(* PLC project Sin nombre, Desconocido Sin nombre 1 *)
(* stored: creationDateTime 2024-11-28T09:53:41, modificationDateTime 2024-12-06T04:11:27 *)

PROGRAM Dimmer
  VAR
    Control_button AT %IX0.0 : BOOL;  (* Push button input *)
    Light_output AT %QX0.0 : BOOL;  (* Light dimmer control output *)
  END_VAR
  VAR
    Light_bright : INT;  (* Step sequence count indicates the bright level *)
    Pulse_regulator : TIME;  (* Value in time of pulse width *)
    Light_on_state : BOOL;  (* Indicates that light is on *)
    Reset_state : BOOL;  (* Reset de counter, change the state to zero *)
    Flag_cicle : BOOL;  (* Flag active during a cicle, 10ms, used to restart *)
    Full_bright : BOOL;  (* Indicates maximum bright, turn the light on directly *)
    CTU0 : CTU;  (* States counter *)
    TP0 : TP;  (* Pulse generator and width corrector *)
    TOF0 : TOF;  (* Cicle generator timer *)
  END_VAR
  VAR  (* added by the conversion: wires and edge detectors of the diagram *)
    R_TRIG1 : R_TRIG;
    R_TRIG2 : R_TRIG;
  END_VAR

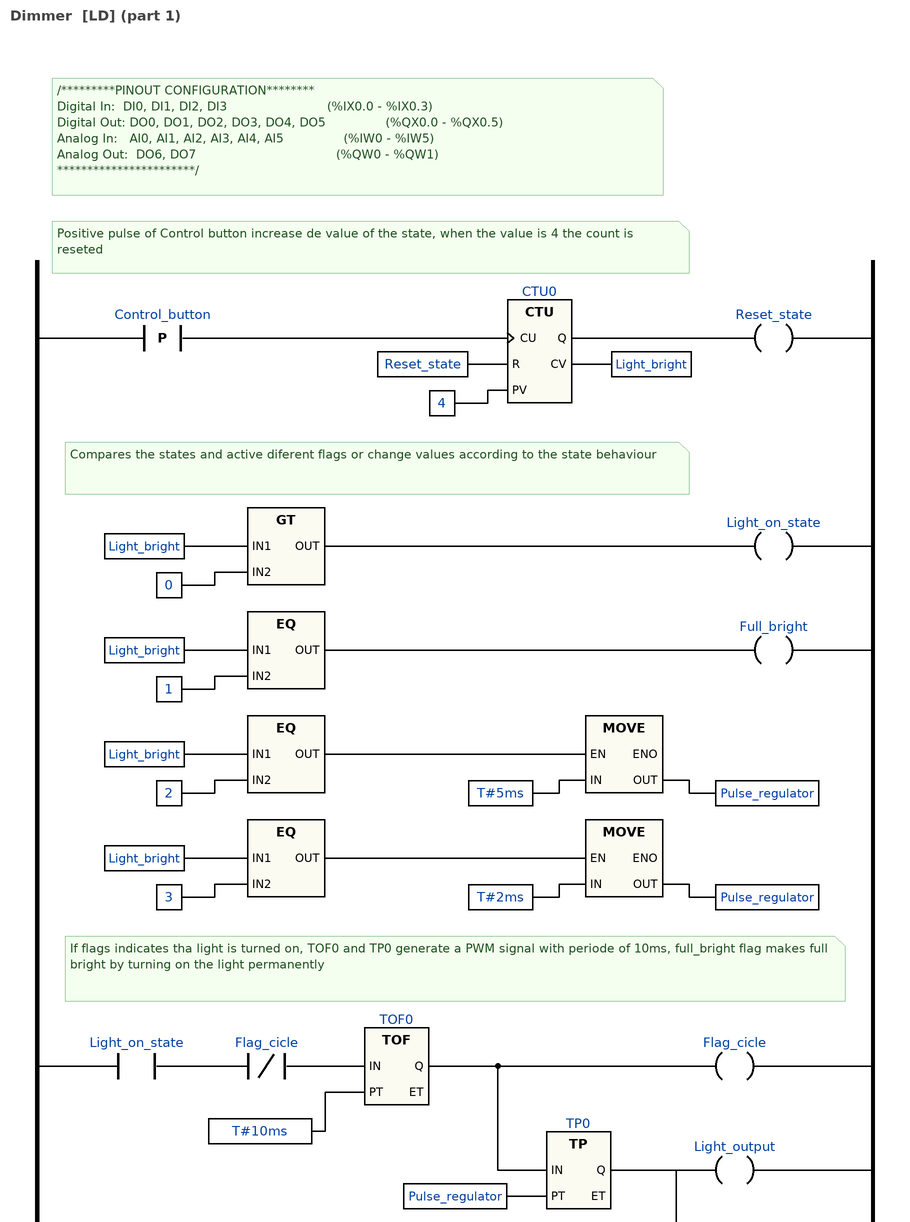
(* LD diagram, written out as Structured Text *)
(* /*********PINOUT CONFIGURATION********
Digital In:  DI0, DI1, DI2, DI3                         (%IX0.0 - %IX0.3)
Digital Out: DO0, DO1, DO2, DO3, DO4, DO5               (%QX0.0 - %QX0.5)
Analog In:   AI0, AI1, AI2, AI3, AI4, AI5               (%IW0 - %IW5)
Analog Out:  DO6, DO7                                   (%QW0 - %QW1)
***********************/ *)
(* Positive pulse of Control button increase de value of the state, when the value is 4 the count is reseted *)
R_TRIG1(CLK := Control_button);
R_TRIG2(CLK := R_TRIG1.Q);
CTU0(CU := R_TRIG2.Q, R := Reset_state, PV := 4);
Reset_state := CTU0.Q;
Light_bright := CTU0.CV;
(* Compares the states and active diferent flags or change values according to the state behaviour *)
(* If flags indicates tha light is turned on, TOF0 and TP0 generate a PWM signal with periode of 10ms, full_bright flag makes full bright by turning on the light permanently *)
TOF0(IN := Light_on_state AND NOT Flag_cicle, PT := T#10ms);
TP0(IN := TOF0.Q, PT := Pulse_regulator);
Light_output := TP0.Q OR Full_bright;
IF Light_bright = 2 THEN Pulse_regulator := T#5ms; END_IF;
IF Light_bright = 3 THEN Pulse_regulator := T#2ms; END_IF;
Flag_cicle := TOF0.Q;
Light_on_state := Light_bright > 0;
Full_bright := Light_bright = 1;
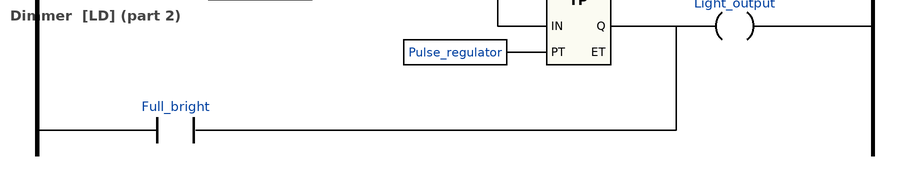
END_PROGRAM

CONFIGURATION Config0
  RESOURCE Res0 ON PLC
    TASK task0(INTERVAL := T#20ms, PRIORITY := 0);
    PROGRAM instance0 WITH task0 : Dimmer;
  END_RESOURCE
END_CONFIGURATION
